PROGRAM treinrit_program
VAR
	Start: BOOL;
	
	 //Timers
	Timer : TON := (PT := gvl.TravelTime);	//train timer

END_VAR

CASE gvl.train OF

0:
IF gvl.bStartTrain AND NOT gvl.InternalStart THEN
	gvl.train := 5;
END_IF;

5:

  	gvl.InternalStart := TRUE;
    gvl.bArrived := FALSE;
    Timer(in := gvl.bStarttrain);
	
IF Timer.Q THEN
    gvl.bArrived := TRUE;
    Timer(IN := FALSE);
    gvl.InternalStart := FALSE;
END_IF;

END_CASE;

END_PROGRAM

(* stored: Version 1.1.0.1, ProductVersion 3.1.4024.15
   POU treinrit_program: Id {6f2205d2-7d14-458c-8068-19fadb977cd2}, SpecialFunc None *)
